TYPE InfoDataAdsAddrStateBase_1916E49F :
STRUCT
END_STRUCT
END_TYPE

(* stored: Version 1.2.0.0, ProductVersion 3.1.4024.9
   DUT InfoDataAdsAddrStateBase_1916E49F: Id {933ea5bc-03b3-4241-aeed-d84d2f2d6eca} *)
